DATA_BLOCK "KukaRobot2_CtrlDB"
{ S7_Optimized_Access := 'FALSE' }
VERSION : 0.1
// ATTRIBUTES
// AUTO_NUMBER = False
// BLOCK_NUMBER = 2402
// END_ATTRIBUTES
"KukaRobot2_Ctrl"

BEGIN

END_DATA_BLOCK

